(* CoDeSys 2.3 library: DOWN_COUNT_TIMER.lib *)
(* Libraries: STANDARD.LIB 5.6.98 11:03:02 *)

(* POU MAIN, LD *)
PROGRAM MAIN
VAR
END_VAR
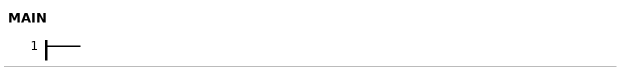
_LD_ (* Ladder Diagram *)
NETWORK 1
	*
_END_LD_
(* the same logic as Structured Text *)
(* Network 1 *)
END_PROGRAM

(* POU DOWN_COUNT_TIMER, LD *)
FUNCTIONBLOCK DOWN_COUNT_TIMER
VAR_INPUT
	BOOL_SIGNAL_IN: BOOL;
	BOOL_TIMER_RST: BOOL;
	INT_AUTO_RST: INT;
	INT_SV_SEC: INT;
END_VAR
VAR_OUTPUT
	SIGNAL_BOOL: BOOL;
	PV_SEC_INT: INT;
END_VAR
VAR
	DF_1: R_TRIG;
	DF_2: R_TRIG;
	M1: BOOL;
	M2: BOOL;

	T100: TON;
	T101: TON;
	M100: BOOL;
	M101: BOOL;
	M200: BOOL;

	M110: BOOL;
	M300: BOOL;
END_VAR
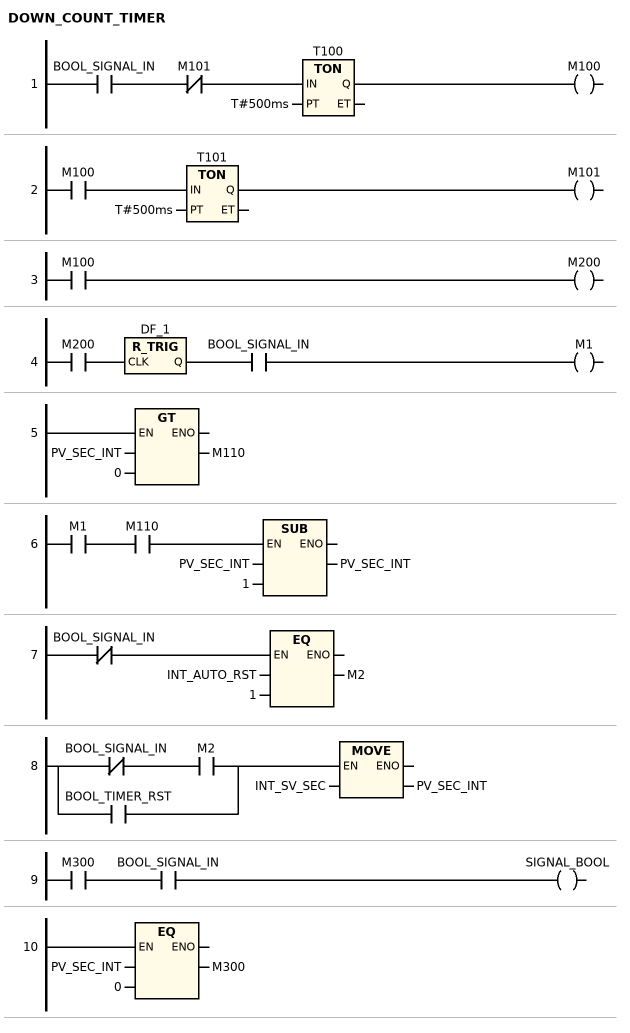
_LD_ (* Ladder Diagram *)
NETWORK 1
	[BOOL_SIGNAL_IN] - [/M101] - T100:TON(IN: *, PT: T#500ms) --- (M100)
NETWORK 2
	[M100] - T101:TON(IN: *, PT: T#500ms) --- (M101)
NETWORK 3
	[M100] --- (M200)
NETWORK 4
	[M200] - DF_1:R_TRIG(CLK: *) - [BOOL_SIGNAL_IN] --- (M1)
NETWORK 5
	*
		EN --- GT(PV_SEC_INT, 0) => M110
NETWORK 6
	[M1] - [M110]
		EN --- SUB(PV_SEC_INT, 1) => PV_SEC_INT
NETWORK 7
	[/BOOL_SIGNAL_IN]
		EN --- EQ(INT_AUTO_RST, 1) => M2
NETWORK 8
	{ [/BOOL_SIGNAL_IN] - [M2] | [BOOL_TIMER_RST] }
		EN --- MOVE(INT_SV_SEC) => PV_SEC_INT
NETWORK 9
	[M300] - [BOOL_SIGNAL_IN] --- (SIGNAL_BOOL)
NETWORK 10
	*
		EN --- EQ(PV_SEC_INT, 0) => M300
_END_LD_
(* the same logic as Structured Text *)
(* Network 1 *)
T100(IN := BOOL_SIGNAL_IN AND NOT M101, PT := T#500ms);
M100 := T100.Q;
(* Network 2 *)
T101(IN := M100, PT := T#500ms);
M101 := T101.Q;
(* Network 3 *)
M200 := M100;
(* Network 4 *)
DF_1(CLK := M200);
M1 := DF_1.Q AND BOOL_SIGNAL_IN;
(* Network 5 *)
M110 := PV_SEC_INT > 0;
(* Network 6 *)
IF M1 AND M110 THEN
	PV_SEC_INT := PV_SEC_INT - 1;
END_IF;
(* Network 7 *)
IF NOT BOOL_SIGNAL_IN THEN
	M2 := INT_AUTO_RST = 1;
END_IF;
(* Network 8 *)
IF NOT BOOL_SIGNAL_IN AND M2 OR BOOL_TIMER_RST THEN
	PV_SEC_INT := INT_SV_SEC;
END_IF;
(* Network 9 *)
SIGNAL_BOOL := M300 AND BOOL_SIGNAL_IN;
(* Network 10 *)
M300 := PV_SEC_INT = 0;
END_FUNCTION_BLOCK
